INTERFACE ITF_Profesor

METHOD Fichar
VAR_INPUT
END_VAR
END_METHOD

PROPERTY Salida : int
GET
END_GET
SET
END_SET
END_PROPERTY

END_INTERFACE

(* stored: Version 1.1.0.1, ProductVersion 3.1.4024.12
   Itf ITF_Profesor: Id {d32aaf3e-2863-41a1-bb8f-9a6473fe3062}
   Method Fichar: Id {8fe518c4-ebed-43e7-b643-f2551c6349ce}
   Property Salida: Id {65cc4ccd-9a72-4d03-be97-7d5471bf5883}
   Get Get: Id {0eaf41a3-232c-4d1a-bab1-51134fe50d76}
   Set Set: Id {df6507f7-5fd9-46a0-aa3d-017dbf527f02} *)
